Yaskawa INFORM job: SBTPOS.JBI

/JOB
//NAME SBTPOS
//POS
///NPOS 0,0,0,0,0,0
//INST
///DATE 2020/09/26 16:07
///ATTR SC,RW,MC
///GROUP1 RB1
///LVARS 4,0,1,0,1,0,0,0
NOP
GETARG LB000 IARG#(1)
GETARG LB001 IARG#(2)
GETARG LB002 IARG#(3)
GETARG LB003 IARG#(4)
SET B070 LB000
SET B071 LB001
SET B072 LB002
SET B073 LB003
SET B069 0
SKILLSND "SpeedbotPos"
WAIT B069=1 T=I010
end
